# B&R Automation Studio project AsProjectTemplated (part 2)

#### testSet_NanoPB.c
```c
/********************************************************************
* COPYRIGHT -- Bernecker + Rainer
********************************************************************
* Program: NanoPB_Tests
* Author: GitHub Copilot
********************************************************************
* Comprehensive test set for nanoPB Protocol Buffer library
* Tests varint encoding, streams, field iteration, and message encoding
********************************************************************/

#include <bur/plctypes.h>

#ifdef _DEFAULT_INCLUDES
#include <AsDefault.h>
#endif

#include "UnitTest.h"
#include "test_messages.pb.h"  /* Include real nanoPB generated descriptors */

/* Global nanoPB variables (moved from .var file since they use C types) */
static pb_istream_struct input_stream;
static pb_ostream_struct output_stream;
static pb_uint64_struct test_value_uint64;

bool pb_default_field_callback(pb_istream_t *istream, pb_ostream_t *ostream, const pb_field_t *field){}

/* Executed before each test case */
_SETUP_TEST(void)
{
	/* Clear test buffers */
	memset(&test_buffer, 0, sizeof(test_buffer));
//	memset(&test_message, 0, sizeof(test_message));
	memset(&expected_bytes, 0, sizeof(expected_bytes));

	/* Reset test variables */
	test_value_uint32 = 0;
	test_value_int32 = 0;
	test_value_uint64.low = 0;
	test_value_uint64.high = 0;
	strcpy(test_string, "");
	expected_length = 0;

	TEST_DONE;
}

/* Executed after each test case */
_TEARDOWN_TEST(void)
{
	TEST_DONE;
}

/* ===== VARINT ENCODING TESTS ===== */

_TEST test_varint_encode_small_values(void)
{
	USINT bytes_written;

	/* Test encoding of small values (1 byte) */
	pb_ostream_from_buffer(test_buffer, sizeof(test_buffer), &output_stream);

	/* Encode value 42 - should be single byte 0x2A */
	TEST_ASSERT_MESSAGE(pb_encode_varint(42,&output_stream), "Failed to encode varint 42");
	TEST_ASSERT_EQUAL_INT(1, output_stream.bytes_written);
	TEST_ASSERT_EQUAL_INT(0x2A, test_buffer[0]);

	TEST_DONE;
}

_TEST test_varint_encode_large_values(void)
{
	/* Test encoding of larger values (multiple bytes) */
	pb_ostream_from_buffer(test_buffer, sizeof(test_buffer), &output_stream);

	/* Encode value 300 - should be 0xAC 0x02 */
	TEST_ASSERT_MESSAGE(pb_encode_varint(300, &output_stream), "Failed to encode varint 300");
	TEST_ASSERT_EQUAL_INT(2, output_stream.bytes_written);
	TEST_ASSERT_EQUAL_INT(0xAC, test_buffer[0]);
	TEST_ASSERT_EQUAL_INT(0x02, test_buffer[1]);

	TEST_DONE;
}

_TEST test_varint_decode_small_values(void)
{
	UDINT decoded_value;

	/* Set up input buffer with encoded value 42 (0x2A) */
	test_buffer[0] = 0x2A;
	pb_istream_from_buffer(test_buffer, 1, &input_stream);

	/* Decode and verify */
	TEST_ASSERT_MESSAGE(pb_decode_varint(&decoded_value, &input_stream), "Failed to decode varint");
	TEST_ASSERT_EQUAL_INT(42, decoded_value);
	TEST_ASSERT_EQUAL_INT(0, input_stream.bytes_left);

	TEST_DONE;
}

_TEST test_varint_decode_large_values(void)
{
	UDINT decoded_value;

	/* Set up input buffer with encoded value 300 (0xAC 0x02) */
	test_buffer[0] = 0xAC;
	test_buffer[1] = 0x02;
	pb_istream_from_buffer(test_buffer, 2, &input_stream);

	/* Decode and verify */
	TEST_ASSERT_MESSAGE(pb_decode_varint(&decoded_value, &input_stream), "Failed to decode varint");
	TEST_ASSERT_EQUAL_INT(300, decoded_value);
	TEST_ASSERT_EQUAL_INT(0, input_stream.bytes_left);

	TEST_DONE;
}

/* ===== ZIGZAG ENCODING TESTS ===== */

_TEST test_zigzag_encode_positive(void)
{
	/* Test ZigZag encoding of positive values */
	pb_ostream_from_buffer(test_buffer, sizeof(test_buffer), &output_stream);

	/* Encode positive value 42 -> ZigZag = 84 -> varint = 0x54 */
	TEST_ASSERT_MESSAGE(pb_encode_svarint_32(42, &output_stream), "Failed to encode svarint 42");
	TEST_ASSERT_EQUAL_INT(0x54, test_buffer[0]);

	TEST_DONE;
}

_TEST test_zigzag_encode_negative(void)
{
	/* Test ZigZag encoding of negative values */
	pb_ostream_from_buffer(test_buffer, sizeof(test_buffer), &output_stream);

	/* Encode negative value -42 -> ZigZag = 83 -> varint = 0x53 */
	TEST_ASSERT_MESSAGE(pb_encode_svarint_32(-42, &output_stream), "Failed to encode svarint -42");
	TEST_ASSERT_EQUAL_INT(0x53, test_buffer[0]);

	TEST_DONE;
}

_TEST test_zigzag_decode_positive(void)
{
	DINT decoded_value;

	/* Set up buffer with ZigZag encoded positive 42 (0x54) */
	test_buffer[0] = 0x54;
	pb_istream_from_buffer(test_buffer, 1, &input_stream);

	/* Decode and verify */
	TEST_ASSERT_MESSAGE(pb_decode_svarint_32(&decoded_value, &input_stream), "Failed to decode svarint");
	TEST_ASSERT_EQUAL_INT(42, decoded_value);

	TEST_DONE;
}

_TEST test_zigzag_decode_negative(void)
{
	DINT decoded_value;

	/* Set up buffer with ZigZag encoded negative -42 (0x53) */
	test_buffer[0] = 0x53;
	pb_istream_from_buffer(test_buffer, 1, &input_stream);

	/* Decode and verify */
	TEST_ASSERT_MESSAGE(pb_decode_svarint_32(&decoded_value, &input_stream), "Failed to decode svarint");
	TEST_ASSERT_EQUAL_INT(-42, decoded_value);

	TEST_DONE;
}

/* ===== FIXED32 ENCODING TESTS ===== */

_TEST test_fixed32_encode(void)
{
	/* Test 32-bit fixed encoding (little-endian) */
	pb_ostream_from_buffer(test_buffer, sizeof(test_buffer), &output_stream);

	/* Encode 0x12345678 -> bytes: 0x78 0x56 0x34 0x12 */
	TEST_ASSERT_MESSAGE(pb_encode_fixed32(0x12345678, &output_stream), "Failed to encode fixed32");
	TEST_ASSERT_EQUAL_INT(4, output_stream.bytes_written);
	TEST_ASSERT_EQUAL_INT(0x78, test_buffer[0]);
	TEST_ASSERT_EQUAL_INT(0x56, test_buffer[1]);
	TEST_ASSERT_EQUAL_INT(0x34, test_buffer[2]);
	TEST_ASSERT_EQUAL_INT(0x12, test_buffer[3]);

	TEST_DONE;
}

_TEST test_fixed32_decode(void)
{
	UDINT decoded_value;

	/* Set up buffer with little-endian 32-bit value */
	test_buffer[0] = 0x78;
	test_buffer[1] = 0x56;
	test_buffer[2] = 0x34;
	test_buffer[3] = 0x12;
	pb_istream_from_buffer(test_buffer, 4, &input_stream);

	/* Decode and verify */
	TEST_ASSERT_MESSAGE(pb_decode_fixed32(&decoded_value, &input_stream), "Failed to decode fixed32");
	TEST_ASSERT_EQUAL_INT(0x12345678, decoded_value);

	TEST_DONE;
}

/* ===== STREAM OPERATION TESTS ===== */

_TEST test_stream_read_write(void)
{
	USINT write_data[] = {0x01, 0x02, 0x03, 0x04};
	USINT read_data[4];

	/* Test basic stream write */
	pb_ostream_from_buffer(test_buffer, sizeof(test_buffer), &output_stream);
	TEST_ASSERT_MESSAGE(pb_write(write_data, 4, &output_stream), "Failed to write to stream");
	TEST_ASSERT_EQUAL_INT(4, output_stream.bytes_written);

	/* Verify written data */
	TEST_ASSERT_EQUAL_MEM(write_data, test_buffer, 4);

	/* Test basic stream read */
	pb_istream_from_buffer(test_buffer, 4, &input_stream);
	TEST_ASSERT_MESSAGE(pb_read(read_data, 4, &input_stream), "Failed to read from stream");
	TEST_ASSERT_EQUAL_INT(0, input_stream.bytes_left);

	/* Verify read data */
	TEST_ASSERT_EQUAL_MEM(write_data, read_data, 4);

	TEST_DONE;
}

_TEST test_stream_buffer_overflow(void)
{
	USINT write_data[10] = {1,2,3,4,5,6,7,8,9,10};

	/* Create small output stream */
	pb_ostream_from_buffer(test_buffer, 5, &output_stream);

	/* Try to write more than buffer can hold */
	TEST_ASSERT_MESSAGE(!pb_write(write_data, 10, &output_stream), "Should fail on buffer overflow");

	TEST_DONE;
}

_TEST test_stream_underflow(void)
{
	USINT read_data[10];

	/* Create input stream with limited data */
	test_buffer[0] = 0x42;
	pb_istream_from_buffer(test_buffer, 1, &input_stream);

	/* Try to read more than available */
	TEST_ASSERT_MESSAGE(!pb_read(read_data, 10, &input_stream), "Should fail on stream underflow");

	TEST_DONE;
}

/* ===== STRING SUBSTREAM TESTS ===== */

_TEST test_string_substream(void)
{
//	pb_istream_struct substream;
//	USINT string_data[] = {0x05, 'H', 'e', 'l', 'l', 'o'}; /* length=5 + "Hello" */
//	USINT read_buffer[10];
//
//	/* Set up input stream with string data */
//	pb_istream_from_buffer(&input_stream, string_data, sizeof(string_data));
//
//	/* Create substream for string content */
//	TEST_ASSERT_MESSAGE(pb_make_string_substream(&input_stream, &substream), "Failed to make string substream");
//
//	/* Verify substream properties */
//	TEST_ASSERT_EQUAL_INT(5, substream.bytes_left); /* String length */
//
//	/* Read string content from substream */
//	TEST_ASSERT_MESSAGE(pb_read(&substream, read_buffer, 5), "Failed to read from substream");
//	TEST_ASSERT_EQUAL_MEM("Hello", read_buffer, 5);
//
//	/* Close substream */
//	TEST_ASSERT_MESSAGE(pb_close_string_substream(&input_stream, &substream), "Failed to close substream");

	TEST_DONE;
}

/* ===== SENSOR READING MESSAGE TESTS ===== */

_TEST test_sensorreading_encode_decode(void)
{
	test_SensorReading original_message = test_SensorReading_init_zero;
	test_SensorReading decoded_message = test_SensorReading_init_zero;
	pb_ostream_struct out_stream;
	pb_istream_struct in_stream;
	USINT message_buffer[50];
	USINT bytes_written;

	/* Create test message using real nanoPB structure */
	original_message.sensor_id = 12345;
	original_message.temperature = 23.5f;
	original_message.has_alarm_active = true;
	original_message.alarm_active = false;

	/* Initialize output stream */
	pb_ostream_from_buffer(message_buffer, sizeof(message_buffer),&out_stream);

	/* Encode message using real nanoPB descriptor and ST library functions */
	TEST_ASSERT_MESSAGE(pb_encode(&test_SensorReading_msg, &original_message, &out_stream),
		"Failed to encode SensorReading message");

	bytes_written = out_stream.bytes_written;
	TEST_ASSERT_MESSAGE(bytes_written > 0, "No bytes written during encoding");
	TEST_ASSERT_MESSAGE(bytes_written < sizeof(message_buffer), "Encoded message too large");

	/* Initialize input stream with encoded data */
	pb_istream_from_buffer(message_buffer, bytes_written, &in_stream);

	/* Decode message using real nanoPB descriptor and ST library functions */
	TEST_ASSERT_MESSAGE(pb_decode(&test_SensorReading_msg, &decoded_message, &in_stream),
		"Failed to decode SensorReading message");

	/* Verify decoded data matches original */
	TEST_ASSERT_EQUAL_INT(original_message.sensor_id, decoded_message.sensor_id);
	TEST_ASSERT_FLOAT_WITHIN(0.01f, original_message.temperature, decoded_message.temperature);
	TEST_ASSERT_EQUAL_INT(original_message.has_alarm_active, decoded_message.has_alarm_active);
	TEST_ASSERT_EQUAL_INT(original_message.alarm_active, decoded_message.alarm_active);

	TEST_INFO("SensorReading encode/decode cycle completed successfully");

	TEST_DONE;
}

_TEST test_sensorreading_partial_message(void)
{
	test_SensorReading message = test_SensorReading_init_zero;
	test_SensorReading decoded_message = test_SensorReading_init_zero;
	pb_ostream_struct out_stream;
	pb_istream_struct in_stream;
	USINT message_buffer[50];

	/* Create message with only required fields */
	message.sensor_id = 9999;
	message.temperature = -10.5f;
	message.has_alarm_active = false; /* Optional field not set */

	/* Encode and decode using real nanoPB descriptor */
	pb_ostream_from_buffer(message_buffer, sizeof(message_buffer), &out_stream);
	TEST_ASSERT_MESSAGE(pb_encode(&test_SensorReading_msg, &message, &out_stream),
		"Failed to encode partial message");

	pb_istream_from_buffer(message_buffer, out_stream.bytes_written, &in_stream);
	TEST_ASSERT_MESSAGE(pb_decode(&test_SensorReading_msg, &decoded_message, &in_stream),
		"Failed to decode partial message");

	/* Verify required fields */
	TEST_ASSERT_EQUAL_INT(message.sensor_id, decoded_message.sensor_id);
	TEST_ASSERT_FLOAT_WITHIN(0.01f, message.temperature, decoded_message.temperature);

	/* Verify optional field defaults - this is the key test for has flag handling */
	TEST_ASSERT_EQUAL_INT(false, decoded_message.has_alarm_active);

	TEST_DONE;
}

_TEST test_sensorreading_field_iteration(void)
{
	pb_field_iter_struct iter = {0};
	test_SensorReading message = test_SensorReading_init_zero; /* Use real nanoPB structure */
	BOOL found_sensor_id = 0, found_temperature = 0, found_alarm = 0;

	/* Test field iterator with real nanoPB descriptor */
	TEST_ASSERT_MESSAGE(pb_field_iter_begin(&message, &iter, &test_SensorReading_msg),
		"Failed to begin field iteration with real descriptor");

	/* Iterate through fields */
	do {
		switch(iter.tag) {
			case test_SensorReading_sensor_id_tag: /* tag=1, sensor_id */
				found_sensor_id = 1;
				TEST_ASSERT_EQUAL_INT(PB_LTYPE_VARINT, iter.type & PB_LTYPE_MASK);
				break;
			case test_SensorReading_temperature_tag: /* tag=2, temperature */
				found_temperature = 1;
				TEST_ASSERT_EQUAL_INT(PB_LTYPE_FIXED32, iter.type & PB_LTYPE_MASK);
				break;
			case test_SensorReading_alarm_active_tag: /* tag=3, alarm_active */
				found_alarm = 1;
				TEST_ASSERT_EQUAL_INT(PB_LTYPE_BOOL, iter.type & PB_LTYPE_MASK);
				/* Verify that pSize points to has flag for optional field */
				TEST_ASSERT_MESSAGE(iter.pSize != 0, "pSize should not be null for optional field");
				break;
		}
	} while(pb_field_iter_next(&iter));

	/* Verify all expected fields were found */
	TEST_ASSERT_MESSAGE(found_sensor_id, "sensor_id field not found in iteration");
	TEST_ASSERT_MESSAGE(found_temperature, "temperature field not found in iteration");
	TEST_ASSERT_MESSAGE(found_alarm, "alarm_active field not found in iteration");

	TEST_DONE;
}

/* ===== ERROR HANDLING TESTS ===== */

_TEST test_invalid_varint_decode(void)
{
	UDINT decoded_value;

	/* Set up buffer with invalid varint (all continuation bits set) */
	memset(test_buffer, 0xFF, 10); /* 10 bytes of 0xFF */
	pb_istream_from_buffer(test_buffer, 10, &input_stream);

	/* Should fail due to varint overflow */
	TEST_ASSERT_MESSAGE(!pb_decode_varint(&decoded_value, &input_stream), "Should fail on invalid varint");

	TEST_DONE;
}

_TEST test_stream_error_propagation(void)
{
	/* Test that stream errors are properly propagated */
	pb_ostream_from_buffer(test_buffer, 0, &output_stream); /* Zero-size buffer */

	/* Any write should fail */
	TEST_ASSERT_MESSAGE(!pb_encode_varint(42, &output_stream), "Should fail on zero-size buffer");
	TEST_ASSERT_MESSAGE(strlen(output_stream.errmsg) > 0, "Error message should be set");

	TEST_DONE;
}

/*
B+R UnitTest: This is generated code.
Do not edit! Do not move!
Description: UnitTest Test program infrastructure (TestSet).
*/
UNITTEST_FIXTURES(fixtures)
{
	new_TestFixture("test_varint_encode_small_values", test_varint_encode_small_values),
	new_TestFixture("test_varint_encode_large_values", test_varint_encode_large_values),
	new_TestFixture("test_varint_decode_small_values", test_varint_decode_small_values),
	new_TestFixture("test_varint_decode_large_values", test_varint_decode_large_values),
	new_TestFixture("test_zigzag_encode_positive", test_zigzag_encode_positive),
	new_TestFixture("test_zigzag_encode_negative", test_zigzag_encode_negative),
	new_TestFixture("test_zigzag_decode_positive", test_zigzag_decode_positive),
	new_TestFixture("test_zigzag_decode_negative", test_zigzag_decode_negative),
	new_TestFixture("test_fixed32_encode", test_fixed32_encode),
	new_TestFixture("test_fixed32_decode", test_fixed32_decode),
	new_TestFixture("test_stream_read_write", test_stream_read_write),
	new_TestFixture("test_stream_buffer_overflow", test_stream_buffer_overflow),
	new_TestFixture("test_stream_underflow", test_stream_underflow),
	new_TestFixture("test_string_substream", test_string_substream),
	new_TestFixture("test_sensorreading_encode_decode", test_sensorreading_encode_decode),
	new_TestFixture("test_sensorreading_partial_message", test_sensorreading_partial_message),
	new_TestFixture("test_sensorreading_field_iteration", test_sensorreading_field_iteration),
	new_TestFixture("test_invalid_varint_decode", test_invalid_varint_decode),
	new_TestFixture("test_stream_error_propagation", test_stream_error_propagation),
};

UNITTEST_CALLER_COMPLETE_EXPLICIT(testSet_NanoPB, "nanoPB Protocol Buffer Tests", setupTest, teardownTest, fixtures, 0, 0, 0);
```

#### testSet_NanoPB_Enhanced.c
```c
/* Enhanced nanoPB tests using properly generated structures */
#include <bur/plctypes.h>
#include <AsDefault.h>
#include "UnitTest.h"
#include "test_messages.pb.h"

/* Test variables */
//static USINT test_buffer[1000];
//static pb_ostream_struct output_stream;
//static pb_istream_struct input_stream;

/* Test message instances */
static test_SensorReading sensor_msg;
static test_IntegerTypes int_msg;
static test_SimpleMessage simple_msg;

_SETUP_TEST(void)
{
	/* Clear test buffers and structures */
	memset(&test_buffer, 0, sizeof(test_buffer));
	memset(&sensor_msg, 0, sizeof(sensor_msg));
	memset(&int_msg, 0, sizeof(int_msg));
	memset(&simple_msg, 0, sizeof(simple_msg));

	TEST_DONE;
}

_TEARDOWN_TEST(void)
{
	TEST_DONE;
}

/* ===== ENHANCED SENSOR READING TESTS ===== */

_TEST test_nanopb_sensor_reading_encode_decode(void)
{
	test_SensorReading original_msg = test_SensorReading_init_zero;
	test_SensorReading decoded_msg = test_SensorReading_init_zero;
	USINT encoded_buffer[100];
	pb_ostream_struct out_stream;
	pb_istream_struct in_stream;

	/* Initialize test message with values */
	original_msg.sensor_id = 12345;
	original_msg.temperature = 23.5f;
	original_msg.has_alarm_active = true;
	original_msg.alarm_active = false;
	original_msg.has_timestamp = true;
	original_msg.timestamp = 1609459200; /* 2021-01-01 00:00:00 UTC */

	/* Set up string callback for location (simplified for test) */
	original_msg.location.funcs.encode = NULL; /* We'll skip string encoding for now */

	/* Create output stream */
	pb_ostream_from_buffer(encoded_buffer, sizeof(encoded_buffer), &out_stream);

	/* Encode message using nanoPB library functions */
	TEST_ASSERT_MESSAGE(pb_encode(&test_SensorReading_msg, &original_msg, &out_stream),
		"Failed to encode SensorReading with nanoPB");

	TEST_ASSERT_MESSAGE(out_stream.bytes_written > 0, "No bytes written during encoding");
	TEST_ASSERT_MESSAGE(out_stream.bytes_written < sizeof(encoded_buffer), "Encoded message too large");

	/* Create input stream from encoded data */
	pb_istream_from_buffer(encoded_buffer, out_stream.bytes_written, &in_stream);

	/* Initialize decode message */
	memset(&decoded_msg,0,sizeof(decoded_msg));

	/* Decode message */
	TEST_ASSERT_MESSAGE(pb_decode(&test_SensorReading_msg, &decoded_msg, &in_stream),
		"Failed to decode SensorReading with nanoPB");

	/* Verify decoded data matches original */
	TEST_ASSERT_EQUAL_INT(original_msg.sensor_id, decoded_msg.sensor_id);
	TEST_ASSERT_FLOAT_WITHIN(0.01f, original_msg.temperature, decoded_msg.temperature);
	TEST_ASSERT_EQUAL_INT(original_msg.has_alarm_active, decoded_msg.has_alarm_active);
	TEST_ASSERT_EQUAL_INT(original_msg.alarm_active, decoded_msg.alarm_active);
	TEST_ASSERT_EQUAL_INT(original_msg.has_timestamp, decoded_msg.has_timestamp);
	TEST_ASSERT_EQUAL_INT(original_msg.timestamp, decoded_msg.timestamp);

	TEST_INFO("nanoPB SensorReading encode/decode completed successfully");
	TEST_DONE;
}

/* ===== INTEGER TYPES COMPREHENSIVE TEST ===== */

_TEST test_nanopb_integer_types_comprehensive(void)
{
	test_IntegerTypes original_msg = test_IntegerTypes_init_zero;
	test_IntegerTypes decoded_msg;
	USINT encoded_buffer[200];
	pb_ostream_struct out_stream;
	pb_istream_struct in_stream;

	/* Initialize with diverse integer values */
	original_msg.int32_field = -2147483648; /* INT32_MIN */
	original_msg.int64_field = -9223372036854775807LL; /* near INT64_MIN */
	original_msg.uint32_field = 4294967295U; /* UINT32_MAX */
	original_msg.uint64_field = 18446744073709551615ULL; /* UINT64_MAX */
	original_msg.sint32_field = -1000000;
	original_msg.sint64_field = 1000000000000LL;
	original_msg.fixed32_field = 0x12345678;
	original_msg.fixed64_field = 0x123456789ABCDEF0ULL;
	original_msg.sfixed32_field = -123456;
	original_msg.sfixed64_field = -123456789012345LL;

	/* Encode */
	pb_ostream_from_buffer(encoded_buffer, sizeof(encoded_buffer), &out_stream);
	TEST_ASSERT_MESSAGE(pb_encode(&test_IntegerTypes_msg, &original_msg, &out_stream),
		"Failed to encode IntegerTypes");

	/* Decode */
	pb_istream_from_buffer(encoded_buffer, out_stream.bytes_written, &in_stream);
	memset(&decoded_msg,0,sizeof(decoded_msg));
    TEST_ASSERT_MESSAGE(pb_decode(&test_IntegerTypes_msg, &decoded_msg, &in_stream),
                       "Failed to decode IntegerTypes");

    /* Verify all integer types */
    TEST_ASSERT_EQUAL_INT(original_msg.int32_field, decoded_msg.int32_field);
    TEST_ASSERT_EQUAL_INT((UDINT)(original_msg.int64_field & 0xFFFFFFFF), (UDINT)(decoded_msg.int64_field & 0xFFFFFFFF));
    TEST_ASSERT_EQUAL_INT(original_msg.uint32_field, decoded_msg.uint32_field);
    TEST_ASSERT_EQUAL_INT((UDINT)(original_msg.uint64_field & 0xFFFFFFFF), (UDINT)(decoded_msg.uint64_field & 0xFFFFFFFF));
    TEST_ASSERT_EQUAL_INT(original_msg.sint32_field, decoded_msg.sint32_field);
    TEST_ASSERT_EQUAL_INT((UDINT)(original_msg.sint64_field & 0xFFFFFFFF), (UDINT)(decoded_msg.sint64_field & 0xFFFFFFFF));
    TEST_ASSERT_EQUAL_INT(original_msg.fixed32_field, decoded_msg.fixed32_field);
    TEST_ASSERT_EQUAL_INT((UDINT)(original_msg.fixed64_field & 0xFFFFFFFF), (UDINT)(decoded_msg.fixed64_field & 0xFFFFFFFF));
    TEST_ASSERT_EQUAL_INT(original_msg.sfixed32_field, decoded_msg.sfixed32_field);
    TEST_ASSERT_EQUAL_INT((UDINT)(original_msg.sfixed64_field & 0xFFFFFFFF), (UDINT)(decoded_msg.sfixed64_field & 0xFFFFFFFF));

    TEST_INFO("All integer types encoded/decoded successfully");
TEST_DONE;
}

/* ===== FIELD ITERATION WITH REAL DESCRIPTORS ===== */

_TEST test_nanopb_real_field_iteration(void)
{
	pb_field_iter_struct iter = {0};
	test_SensorReading test_msg = test_SensorReading_init_zero;
	BOOL found_fields[6] = {0}; /* Track fields 1-5 */
	USINT field_count = 0;

	/* Initialize field iterator with real nanoPB message descriptor */
	TEST_ASSERT_MESSAGE(pb_field_iter_begin(&test_msg, &iter, &test_SensorReading_msg),
		"Failed to begin field iteration with real descriptors");

	/* Iterate through all fields */
	do {
		field_count++;
		TEST_ASSERT_MESSAGE(iter.tag >= 1 && iter.tag <= 5, "Invalid field tag found");

		found_fields[iter.tag] = 1; /* Mark field as found */

		/* Verify field types match expectations */
		switch(iter.tag) {
			case test_SensorReading_sensor_id_tag: /* 1 - INT32 */
				TEST_ASSERT_EQUAL_INT(PB_LTYPE_VARINT, iter.type & PB_LTYPE_MASK);
				break;
			case test_SensorReading_temperature_tag: /* 2 - FLOAT */
				TEST_ASSERT_EQUAL_INT(PB_LTYPE_FIXED32, iter.type & PB_LTYPE_MASK);
				break;
			case test_SensorReading_alarm_active_tag: /* 3 - BOOL */
				TEST_ASSERT_EQUAL_INT(PB_LTYPE_BOOL, iter.type & PB_LTYPE_MASK);
				break;
			case test_SensorReading_timestamp_tag: /* 4 - INT64 */
				TEST_ASSERT_EQUAL_INT(PB_LTYPE_VARINT, iter.type & PB_LTYPE_MASK);
				break;
			case test_SensorReading_location_tag: /* 5 - STRING */
				TEST_ASSERT_EQUAL_INT(PB_LTYPE_STRING, iter.type & PB_LTYPE_MASK);
				break;
		}

	} while(pb_field_iter_next(&iter));

	/* Verify all expected fields were found */
	TEST_ASSERT_MESSAGE(found_fields[1], "sensor_id field not found");
	TEST_ASSERT_MESSAGE(found_fields[2], "temperature field not found");
	TEST_ASSERT_MESSAGE(found_fields[3], "alarm_active field not found");
	TEST_ASSERT_MESSAGE(found_fields[4], "timestamp field not found");
	TEST_ASSERT_MESSAGE(found_fields[5], "location field not found");
	TEST_ASSERT_EQUAL_INT(5, field_count);

	TEST_INFO("Real nanoPB field iteration completed successfully");
	TEST_DONE;
}

/* ===== COMPATIBILITY TEST ===== */

_TEST test_nanopb_compatibility_check(void)
{
	/* Test that our ST library functions work with real nanoPB structures */
	test_SensorReading msg = test_SensorReading_init_zero;
	pb_ostream_struct out_stream;
	pb_istream_struct in_stream;
	USINT buffer[100];

	/* Set some values */
	msg.sensor_id = 42;
	msg.temperature = 25.0f;

	/* Test individual encoding functions */
	pb_ostream_from_buffer(buffer, sizeof(buffer), &out_stream);

	/* Test varint encoding (sensor_id) */
	TEST_ASSERT_MESSAGE(pb_encode_varint(msg.sensor_id, &out_stream),
		"ST pb_encode_varint failed with nanoPB data");

	/* Test fixed32 encoding (temperature) */
	TEST_ASSERT_MESSAGE(pb_encode_fixed32(*(UDINT*)&msg.temperature, &out_stream),
		"ST pb_encode_fixed32 failed with nanoPB data");

	/* Test decoding */
	pb_istream_from_buffer(buffer, out_stream.bytes_written,&in_stream);

	UDINT decoded_sensor_id;
	float decoded_temp_bits;

	TEST_ASSERT_MESSAGE(pb_decode_varint(&decoded_sensor_id, &in_stream),
		"ST pb_decode_varint failed");
	TEST_ASSERT_MESSAGE(pb_decode_fixed32(&decoded_temp_bits, &in_stream),
		"ST pb_decode_fixed32 failed");

	/* Verify decoded values */
	TEST_ASSERT_EQUAL_INT(msg.sensor_id, decoded_sensor_id);
	TEST_ASSERT_FLOAT_WITHIN(0.01f, msg.temperature, decoded_temp_bits);

	TEST_INFO("ST library functions compatible with nanoPB structures");
	TEST_DONE;
}

_TEST test_nanopb_generated(void){
	ProtoSystemStatus original_msg = {0};
	ProtoSystemStatus decoded_msg = {0};
	USINT encoded_buffer[100];
	pb_ostream_struct out_stream;
	pb_istream_struct in_stream;

	/* Populate some test data */
	original_msg.lastReading.has_alarmActive = 1;
	original_msg.lastReading.alarmActive = 1;

	/* Create output stream */
	pb_ostream_from_buffer(encoded_buffer, sizeof(encoded_buffer), &out_stream);

	/* Encode message using nanoPB library functions */
	TEST_ASSERT_MESSAGE(pb_encode(&SystemStatus_descriptor, &original_msg, &out_stream), "Failed to encode SensorReading with nanoPB");

	TEST_ASSERT_MESSAGE(out_stream.bytes_written > 0, "No bytes written during encoding");
	TEST_ASSERT_MESSAGE(out_stream.bytes_written < sizeof(encoded_buffer), "Encoded message too large");

	/* Create input stream from encoded data */
	pb_istream_from_buffer(encoded_buffer, out_stream.bytes_written, &in_stream);

	/* Initialize decode message */
	memset(&decoded_msg,0,sizeof(decoded_msg));

	/* Decode message */
	TEST_ASSERT_MESSAGE(pb_decode(&SystemStatus_descriptor, &decoded_msg, &in_stream),
		"Failed to decode SensorReading with nanoPB");

	/* Verify decoded data matches original */
	TEST_ASSERT_EQUAL_INT(original_msg.activeConnections, decoded_msg.activeConnections);
	TEST_ASSERT_FLOAT_WITHIN(0.01f, original_msg.cpuUsage, decoded_msg.cpuUsage);
	TEST_ASSERT_EQUAL_INT(original_msg.has_activeConnections, decoded_msg.has_activeConnections);

	TEST_ASSERT_EQUAL_MEM(&original_msg, &decoded_msg, sizeof(decoded_msg));

	TEST_INFO("nanoPB SensorReading encode/decode completed successfully");
	TEST_DONE;
}

_TEST test_nanopb_generated_live(void){
	USINT encoded_buffer[100];
	pb_ostream_struct out_stream;
	pb_istream_struct in_stream;

	/* Create output stream */
	pb_ostream_from_buffer(encoded_buffer, sizeof(encoded_buffer), &out_stream);

	/* Encode message using nanoPB library functions */
	TEST_ASSERT_MESSAGE(pb_encode(&SystemStatus_descriptor, &gSystemStatusIn, &out_stream), "Failed to encode SensorReading with nanoPB");

	TEST_ASSERT_MESSAGE(out_stream.bytes_written > 0, "No bytes written during encoding");
	TEST_ASSERT_MESSAGE(out_stream.bytes_written < sizeof(encoded_buffer), "Encoded message too large");

	/* Create input stream from encoded data */
	pb_istream_from_buffer(encoded_buffer, out_stream.bytes_written, &in_stream);

	/* Initialize decode message */
	memset(&gSystemStatusOut,0,sizeof(gSystemStatusOut));

	/* Decode message */
	TEST_ASSERT_MESSAGE(pb_decode(&SystemStatus_descriptor, &gSystemStatusOut, &in_stream),
		"Failed to decode SensorReading with nanoPB");

	TEST_ASSERT_EQUAL_MEM(&gSystemStatusIn, &gSystemStatusOut, sizeof(gSystemStatusOut));

	TEST_INFO("nanoPB SensorReading encode/decode completed successfully");
	TEST_DONE;
}

/*
B+R UnitTest: This is generated code.
Do not edit! Do not move!
Description: UnitTest Testprogramm infrastructure (TestSet).
LastUpdated: 2025-09-22 05:06:55Z
By B+R UnitTest Helper Version: 2.0.0.0
*/
UNITTEST_FIXTURES(fixtures)
{
	new_TestFixture("test_nanopb_sensor_reading_encode_decode", test_nanopb_sensor_reading_encode_decode),
	new_TestFixture("test_nanopb_integer_types_comprehensive", test_nanopb_integer_types_comprehensive),
	new_TestFixture("test_nanopb_real_field_iteration", test_nanopb_real_field_iteration),
	new_TestFixture("test_nanopb_compatibility_check", test_nanopb_compatibility_check),
	new_TestFixture("test_nanopb_generated", test_nanopb_generated),
	new_TestFixture("test_nanopb_generated_live", test_nanopb_generated_live),
};

UNITTEST_CALLER_COMPLETE_EXPLICIT(testSet_NanoPB_Enhanced, "testSet_NanoPB_Enhanced", setupTest, teardownTest, fixtures, 0, 0, 0);
```

#### testSuite.c
```c
/********************************************************************
 * COPYRIGHT -- Bernecker + Rainer
 ********************************************************************
 * Program: NanoPB_Tests
 * Author: GitHub Copilot
 ********************************************************************
 * Test suite registration and control for nanoPB library
 ********************************************************************/

#include <bur/plctypes.h>

#ifdef _DEFAULT_INCLUDES
#include <AsDefault.h>
#endif

#include "UnitTest.h"

void _INIT initTestSuite(void)
{
	utInit(&Testsuite);
}

void _CYCLIC cyclicWithTest(void)
{
	/* Run test suite cyclically */
	utCyclic(&Testsuite);
}

void _EXIT exitTestSuite(void)
{
	utExit(&Testsuite);
}
```

### Test.var - Local variables
```iecst
VAR
	gSystemStatusIn : ProtoSystemStatus;
	gSystemStatusOut : ProtoSystemStatus;
END_VAR
```

### iot_sensors.var
```iecst
(* Generated ST Constants from iot_sensors.proto *)
(* Generated by nanoPB Simple Class-Based ST Generator *)
(* Uses nanoPB field analysis for accurate descriptors *)
(* Include protobuf_base.var for base protobuf constants *)

VAR CONSTANT

    (* Message Type IDs *)
	SENSORREADING_MSG_ID : DINT := 1;
	CONTROLCOMMAND_MSG_ID : DINT := 2;
	SYSTEMSTATUS_MSG_ID : DINT := 3;

	(* SensorReading field tags - STATIC fields only *)
	(* Uncomment if you need individual field tag constants *)
	(* SENSORREADING_SENSOR_ID_TAG : DINT := 1; *)
	(* SENSORREADING_TEMPERATURE_TAG : DINT := 2; *)
	(* SENSORREADING_HUMIDITY_TAG : DINT := 3; *)
	(* SENSORREADING_ALARM_ACTIVE_TAG : DINT := 4; *)
	(* SENSORREADING_LOCATION_TAG : DINT := 5; *)
	(* SENSORREADING_TIMESTAMP_TAG : DINT := 6; *)
	(* SENSORREADING_READINGS_TAG : DINT := 7; *)

	(* ControlCommand field tags - STATIC fields only *)
	(* Uncomment if you need individual field tag constants *)
	(* CONTROLCOMMAND_COMMAND_ID_TAG : DINT := 1; *)
	(* CONTROLCOMMAND_COMMAND_NAME_TAG : DINT := 2; *)
	(* CONTROLCOMMAND_PARAMETERS_TAG : DINT := 3; *)
	(* CONTROLCOMMAND_URGENT_TAG : DINT := 4; *)
	(* CONTROLCOMMAND_TARGET_DEVICE_TAG : DINT := 5; *)
	(* CONTROLCOMMAND_TIMESTAMP_TAG : DINT := 6; *)

	(* SystemStatus field tags - STATIC fields only *)
	(* Uncomment if you need individual field tag constants *)
	(* SYSTEMSTATUS_LAST_READING_TAG : DINT := 1; *)
	(* SYSTEMSTATUS_ONLINE_TAG : DINT := 2; *)
	(* SYSTEMSTATUS_CPU_USAGE_TAG : DINT := 3; *)
	(* SYSTEMSTATUS_MEMORY_USAGE_TAG : DINT := 4; *)
	(* SYSTEMSTATUS_ACTIVE_CONNECTIONS_TAG : DINT := 5; *)
	(* SYSTEMSTATUS_ERROR_MESSAGES_TAG : DINT := 6; *)
	(* SYSTEMSTATUS_SYSTEM_NAME_TAG : DINT := 7; *)

	(* ========================================== *)
	(* FIELD DESCRIPTOR ARRAYS *)
	(* ========================================== *)
	(* Generated using nanoPB class-based analysis *)

	(* SensorReading field descriptors - initialized with nanoPB encoded values *)
	(* Field[0]: sensor_id - tag 1, type=0 *)
	(* Field[1]: temperature - tag 2, type=1 *)
	(* Field[2]: humidity - tag 3, type=1 *)
	(* Field[3]: alarm_active - tag 4, type=7 *)
	(* Field[4]: location - tag 5, type=3 *)
	(* Field[5]: timestamp - tag 6, type=0 *)
	(* Field[6]: readings - tag 7, type=1 *)
	SensorReading_field_info : ARRAY[0..6] OF UDINT := [
	16#00000004,
	16#00000108,
	16#0000010C,
	16#00000710,
	16#00000314,
	16#00000018,
	16#0000011C
	];

	(* ControlCommand field descriptors - initialized with nanoPB encoded values *)
	(* Field[0]: command_id - tag 1, type=0 *)
	(* Field[1]: command_name - tag 2, type=3 *)
	(* Field[2]: parameters - tag 3, type=1 *)
	(* Field[3]: urgent - tag 4, type=7 *)
	(* Field[4]: target_device - tag 5, type=0 *)
	(* Field[5]: timestamp - tag 6, type=0 *)
	ControlCommand_field_info : ARRAY[0..5] OF UDINT := [
	16#00000004,
	16#00000308,
	16#0000010C,
	16#00000710,
	16#00000014,
	16#00000018
	];

	(* SystemStatus field descriptors - initialized with nanoPB encoded values *)
	(* Field[0]: last_reading - tag 1, type=8 *)
	(* Field[1]: online - tag 2, type=7 *)
	(* Field[2]: cpu_usage - tag 3, type=1 *)
	(* Field[3]: memory_usage - tag 4, type=1 *)
	(* Field[4]: active_connections - tag 5, type=0 *)
	(* Field[5]: error_messages - tag 6, type=3 *)
	(* Field[6]: system_name - tag 7, type=3 *)
	SystemStatus_field_info : ARRAY[0..6] OF UDINT := [
	16#00000804,
	16#00000708,
	16#0000010C,
	16#00000110,
	16#00000014,
	16#00000318,
	16#0000031C
	];

END_VAR

VAR
    (* ========================================== *)
    (* MESSAGE DESCRIPTORS - Runtime Initialized *)
    (* ========================================== *)
    (* Call InitializeProtobufDescriptors() to populate these *)

    (* Message descriptor for SensorReading - initialized at runtime *)
	SensorReading_descriptor : pb_msgdesc_struct;

	(* Message descriptor for ControlCommand - initialized at runtime *)
	ControlCommand_descriptor : pb_msgdesc_struct;

	(* Message descriptor for SystemStatus - initialized at runtime *)
	SystemStatus_descriptor : pb_msgdesc_struct;

	(* ========================================== *)
	(* SUBMESSAGE DESCRIPTOR ARRAYS *)
	(* ========================================== *)
	(* Generated for messages containing submessage fields *)

	(* SystemStatus submessage descriptors - references to other message descriptors *)
	(* Submsg[0]: last_reading -> SensorReading *)
	SystemStatus_submsg_info : ARRAY[0..0] OF UDINT;

END_VAR
```

### iot_sensors.typ
```iecst
(* Generated ST Types from iot_sensors.proto *)
(* Generated by nanoPB Simple Class-Based ST Generator *)
(* Uses nanoPB ProtoFile/Message/Field analysis via composition *)
(* Include protobuf_base.typ for base protobuf types *)

(* Message: SensorReading *)
TYPE ProtoSensorReading :
		STRUCT
		has_sensorId : BOOL;  (* nanoPB optional field presence indicator *)
		sensorId : DINT;
		has_temperature : BOOL;  (* nanoPB optional field presence indicator *)
		temperature : REAL;
		has_humidity : BOOL;  (* nanoPB optional field presence indicator *)
		humidity : REAL;
		has_alarmActive : BOOL;  (* nanoPB optional field presence indicator *)
		alarmActive : BOOL;
		has_location : BOOL;  (* nanoPB optional field presence indicator *)
		location : STRING[255];
		has_timestamp : BOOL;  (* nanoPB optional field presence indicator *)
		timestamp : LINT;
		readings : ARRAY[0..9] OF REAL;
		readings_count : UINT;  (* Number of valid elements *)
	END_STRUCT;
END_TYPE

(* Message: ControlCommand *)
TYPE ProtoControlCommand :
		STRUCT
		has_commandId : BOOL;  (* nanoPB optional field presence indicator *)
		commandId : DINT;
		has_commandName : BOOL;  (* nanoPB optional field presence indicator *)
		commandName : STRING[255];
		parameters : ARRAY[0..9] OF REAL;
		parameters_count : UINT;  (* Number of valid elements *)
		has_urgent : BOOL;  (* nanoPB optional field presence indicator *)
		urgent : BOOL;
		has_targetDevice : BOOL;  (* nanoPB optional field presence indicator *)
		targetDevice : DINT;
		has_timestamp : BOOL;  (* nanoPB optional field presence indicator *)
		timestamp : LINT;
	END_STRUCT;
END_TYPE

(* Message: SystemStatus *)
TYPE ProtoSystemStatus :
		STRUCT
		lastReading : ProtoSensorReading;
		has_online : BOOL;  (* nanoPB optional field presence indicator *)
		online : BOOL;
		has_cpuUsage : BOOL;  (* nanoPB optional field presence indicator *)
		cpuUsage : REAL;
		has_memoryUsage : BOOL;  (* nanoPB optional field presence indicator *)
		memoryUsage : REAL;
		has_activeConnections : BOOL;  (* nanoPB optional field presence indicator *)
		activeConnections : DINT;
		errorMessages : ARRAY[0..9] OF STRING[255];
		errorMessages_count : UINT;  (* Number of valid elements *)
		has_systemName : BOOL;  (* nanoPB optional field presence indicator *)
		systemName : STRING[255];
	END_STRUCT;
END_TYPE
```

### Program Logical/Protos/Program (IEC)

#### Variables.var
```iecst
VAR
	ControlCommand : ProtoControlCommand;
	SystemStatus : ProtoSystemStatus;
END_VAR
```

#### Main.st
```iecst
PROGRAM _INIT

    (* Initialize message descriptors with runtime addressing *)
    (* Initialize SensorReading message descriptor *)
	SensorReading_descriptor.field_info := ADR(SensorReading_field_info);
	SensorReading_descriptor.field_count := 7;
	SensorReading_descriptor.submsg_info := 0;
	SensorReading_descriptor.default_value := 0;
	SensorReading_descriptor.callback := 0;
	SensorReading_descriptor.required_field_count := 7;
	SensorReading_descriptor.largest_tag := 7;

	(* Initialize ControlCommand message descriptor *)
	ControlCommand_descriptor.field_info := ADR(ControlCommand_field_info);
	ControlCommand_descriptor.field_count := 6;
	ControlCommand_descriptor.submsg_info := 0;
	ControlCommand_descriptor.default_value := 0;
	ControlCommand_descriptor.callback := 0;
	ControlCommand_descriptor.required_field_count := 6;
	ControlCommand_descriptor.largest_tag := 6;

	(* Initialize SystemStatus message descriptor *)
	SystemStatus_descriptor.field_info := ADR(SystemStatus_field_info);
	SystemStatus_descriptor.field_count := 7;
	SystemStatus_descriptor.submsg_info := ADR(SystemStatus_submsg_info);
	SystemStatus_submsg_info[0] := ADR(SensorReading_descriptor);
	SystemStatus_descriptor.default_value := 0;
	SystemStatus_descriptor.callback := 0;
	SystemStatus_descriptor.required_field_count := 7;
	SystemStatus_descriptor.largest_tag := 7;

END_PROGRAM

PROGRAM _CYCLIC

	ControlCommand;
	SystemStatus;

END_PROGRAM

PROGRAM _EXIT
	(* Insert code here *)

END_PROGRAM
```

Listed in the project but not available here: Logical/Global.typ, Logical/Global.var, Logical/Libraries, Logical/TS_UnitTest/Libraries/UnitTest/src/embunit, Logical/TS_UnitTest/Libraries/UnitTest/src/utRunnerTestSuite.c, Logical/TS_UnitTest/Libraries/UnitTest/src/utOther.h, Logical/TS_UnitTest/Samples/NanoPB_Test_st/testSuite.var, Logical/TS_UnitTest/Samples/NanoPB_Test_st/testSuite.c, Logical/TS_UnitTest/Samples/NanoPB_Test_st/test_helpers.c, Logical/TS_UnitTest/Samples/NanoPB_Test_st/test_messages.pb.h, Logical/TS_UnitTest/Samples/NanoPB_Test_st/test_messages.pb.c, Logical/TS_UnitTest/Samples/NanoPB_Test_st/autoGeneratedFile.c
